INTERFACE ITF_Component EXTENDS ITF_BaseComponent

END_INTERFACE

(* stored: Version 1.1.0.1, ProductVersion 3.1.4024.15
   Itf ITF_Component: Id {049be64b-6a97-47c2-87b8-7adecc4d1d51} *)
